// TwinCAT 3 PLC project Plc
// ProgramVersion: 3.1.4024.0
// libraries:
//   Tc2_Standard, * (Beckhoff Automation GmbH)
//   Tc2_System, * (Beckhoff Automation GmbH)
//   Tc3_Module, * (Beckhoff Automation GmbH)
//   VisuDialogs, * (System)
// project tree:
//   / Gestore di visualizzazione.TcVMO (not stored), GlobalTextList.TcGTLO, ImagePool.TcIPO (not stored), PlcTask.TcTTO, VisuTask.TcTTO
//   GVLs/ GVL.TcGVL (not stored)
//   POUs/ MAIN.TcPOU, VISU.TcPOU
//   VISUs/ Visualization.TcVIS
// real-time tasks:
//   TASK PlcTask: cycle T#10ms, priority 20, ADS port 350
//   TASK VisuTask: cycle T#100000us, priority 60, ADS port 351

CONFIGURATION Plc
    RESOURCE PLC ON TwinCAT3
        TASK PlcTask(INTERVAL := T#10ms, PRIORITY := 20);
        TASK VisuTask(INTERVAL := T#100000us, PRIORITY := 60);
        PROGRAM MAIN WITH PlcTask : MAIN;
    END_RESOURCE
END_CONFIGURATION

// ---- POUs/MAIN.TcPOU
PROGRAM MAIN
VAR
	StopRichiesto: BOOL;
	Anomalia: BOOL;
	Emergenza: BOOL;
	Funzione: BOOL;
	Smistamento: BOOL;
	Rotazione: BOOL;
	AttivaMicroRulli: BOOL;
	FineSmistamento: BOOL;
	FinePesatura: BOOL;
	RuotaOrigine: BOOL;
	PesoMin5: BOOL;
	PesoMag10: BOOL;
	PesoIntermedio: BOOL;
	ProsciuttoSmistato: BOOL;
	ProsciuttiTotali: UINT;
	ProsciuttiCommerciabili: UINT;
	PercentualeProsciuttiCommerciabili: UINT;
	//Timer
	TON_PS1: TON;
	TON_Pesatura: TON;
	TON_MicroRulli: TON;
	TON_Min5: TON;
	TON_Mag10: TON;
	TON_Intermedi: TON;
	//Counter
	CTU_Min5: CTU;
	CTU_Mag10: CTU;
	CTU_Intermedi: CTU;
END_VAR

GestionePulsanti();
GestioneMotori();
GestionePesatura();
GestioneRotazione();
GestioneSmistamento();
GestioneConteggio();

ACTION GestioneConteggio:
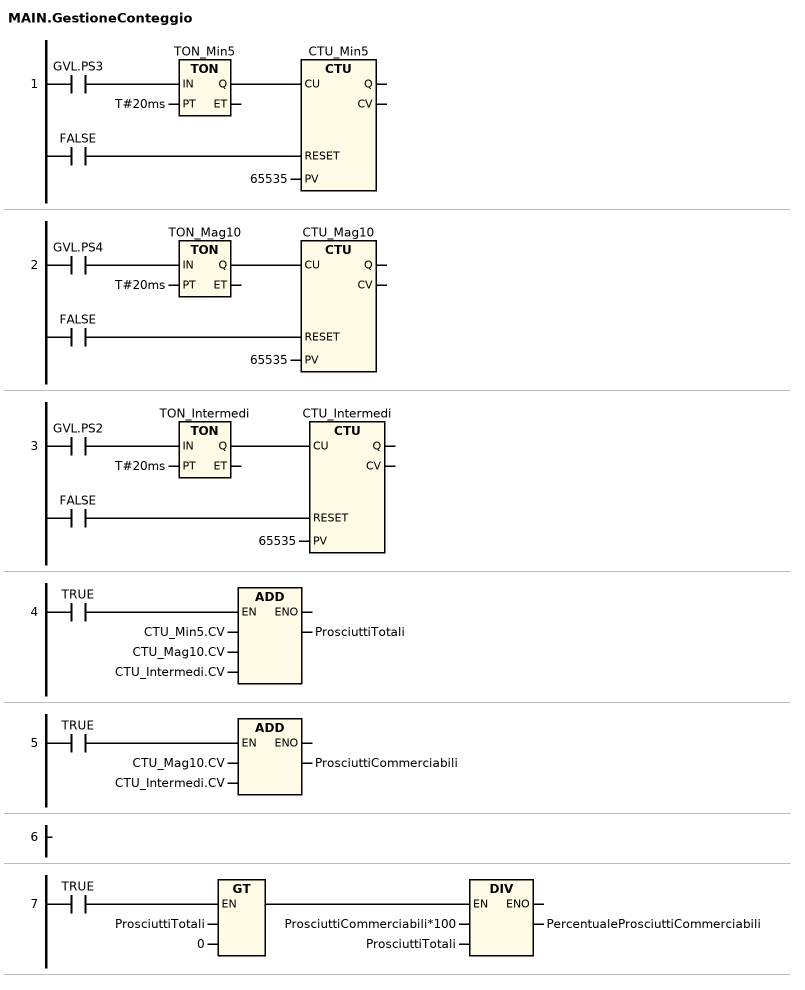
// NETWORK 1
TON_Min5(IN := GVL.PS3, PT := T#20ms); // TON
CTU_Min5(CU := TON_Min5.Q, RESET := FALSE, PV := 65535); // CTU

// NETWORK 2
TON_Mag10(IN := GVL.PS4, PT := T#20ms); // TON
CTU_Mag10(CU := TON_Mag10.Q, RESET := FALSE, PV := 65535); // CTU

// NETWORK 3
TON_Intermedi(IN := GVL.PS2, PT := T#20ms); // TON
CTU_Intermedi(CU := TON_Intermedi.Q, RESET := FALSE, PV := 65535); // CTU

// NETWORK 4
ProsciuttiTotali := CTU_Min5.CV + CTU_Mag10.CV + CTU_Intermedi.CV;

// NETWORK 5
ProsciuttiCommerciabili := CTU_Mag10.CV + CTU_Intermedi.CV;

// NETWORK 6

// NETWORK 7
IF ProsciuttiTotali > 0 THEN
    PercentualeProsciuttiCommerciabili := (ProsciuttiCommerciabili*100) / ProsciuttiTotali;
END_IF
END_ACTION

ACTION GestioneMotori:
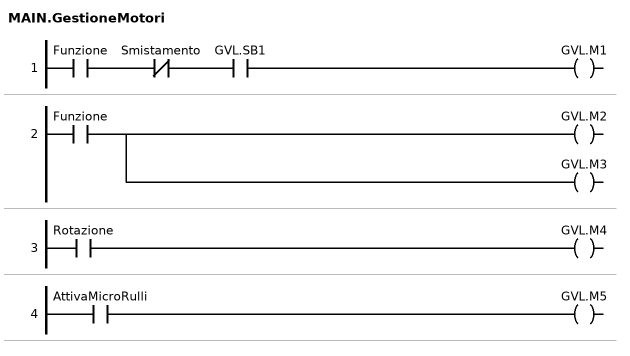
// NETWORK 1
GVL.M1 := Funzione AND NOT Smistamento AND GVL.SB1;

// NETWORK 2
GVL.M2 := Funzione;
GVL.M3 := Funzione;

// NETWORK 3
GVL.M4 := Rotazione;

// NETWORK 4
GVL.M5 := AttivaMicroRulli;
END_ACTION

ACTION GestionePesatura:
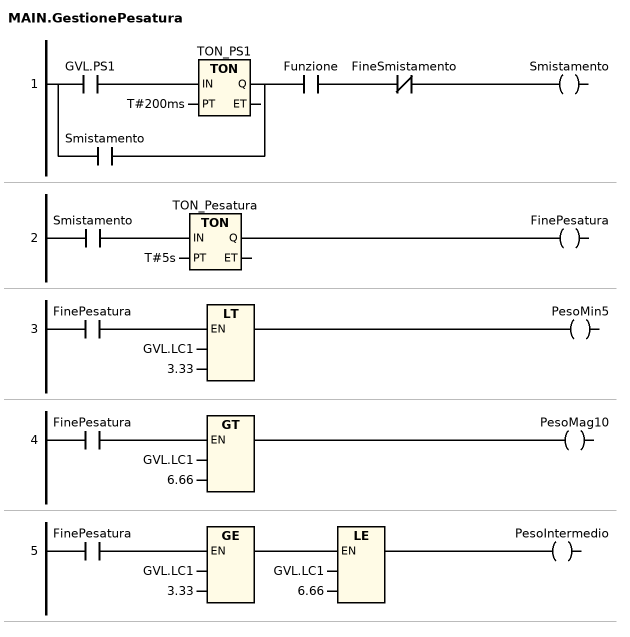
// NETWORK 1
TON_PS1(IN := GVL.PS1, PT := T#200ms); // TON
Smistamento := (TON_PS1.Q OR Smistamento) AND Funzione AND NOT FineSmistamento;

// NETWORK 2
TON_Pesatura(IN := Smistamento, PT := T#5s); // TON
FinePesatura := TON_Pesatura.Q;

// NETWORK 3
PesoMin5 := FinePesatura AND GVL.LC1 < 3.33;

// NETWORK 4
PesoMag10 := FinePesatura AND GVL.LC1 > 6.66;

// NETWORK 5
PesoIntermedio := FinePesatura AND GVL.LC1 >= 3.33 AND GVL.LC1 <= 6.66;
END_ACTION

ACTION GestionePulsanti:
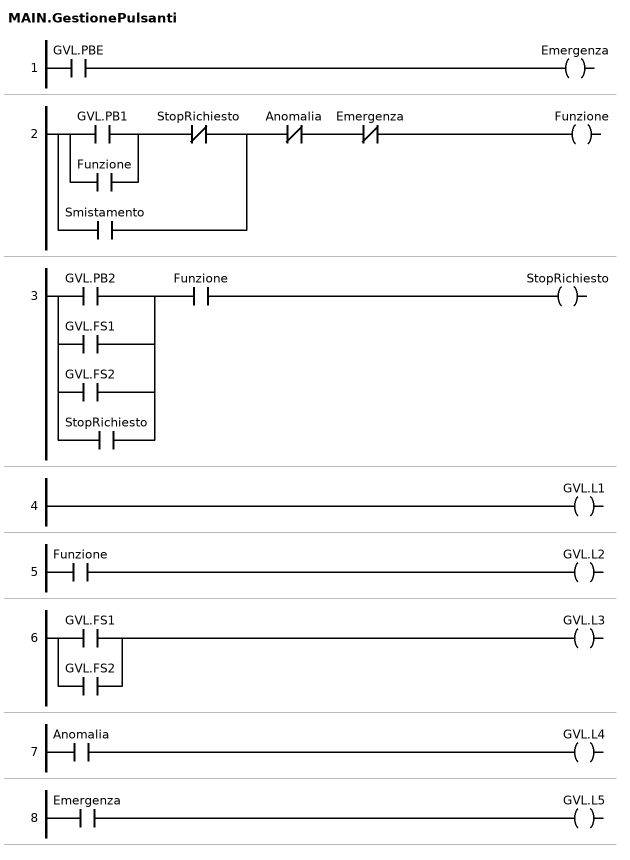
// NETWORK 1
Emergenza := GVL.PBE;

// NETWORK 2
Funzione := ((GVL.PB1 OR Funzione) AND NOT StopRichiesto OR Smistamento) AND NOT Anomalia AND NOT Emergenza;

// NETWORK 3
StopRichiesto := (GVL.PB2 OR GVL.FS1 OR GVL.FS2 OR StopRichiesto) AND Funzione;

// NETWORK 4
GVL.L1 := TRUE;

// NETWORK 5
GVL.L2 := Funzione;

// NETWORK 6
GVL.L3 := GVL.FS1 OR GVL.FS2;

// NETWORK 7
GVL.L4 := Anomalia;

// NETWORK 8
GVL.L5 := Emergenza;
END_ACTION

ACTION GestioneRotazione:
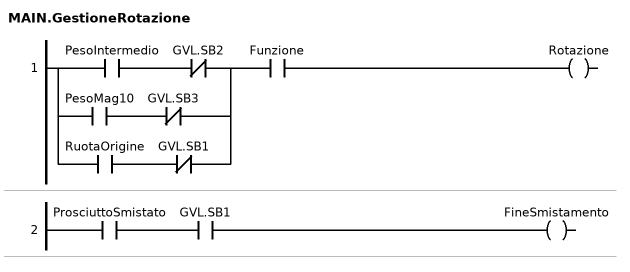
// NETWORK 1
Rotazione := (PesoIntermedio AND NOT GVL.SB2 OR PesoMag10 AND NOT GVL.SB3 OR RuotaOrigine AND NOT GVL.SB1) AND Funzione;

// NETWORK 2
FineSmistamento := ProsciuttoSmistato AND GVL.SB1;
END_ACTION

ACTION GestioneSmistamento:
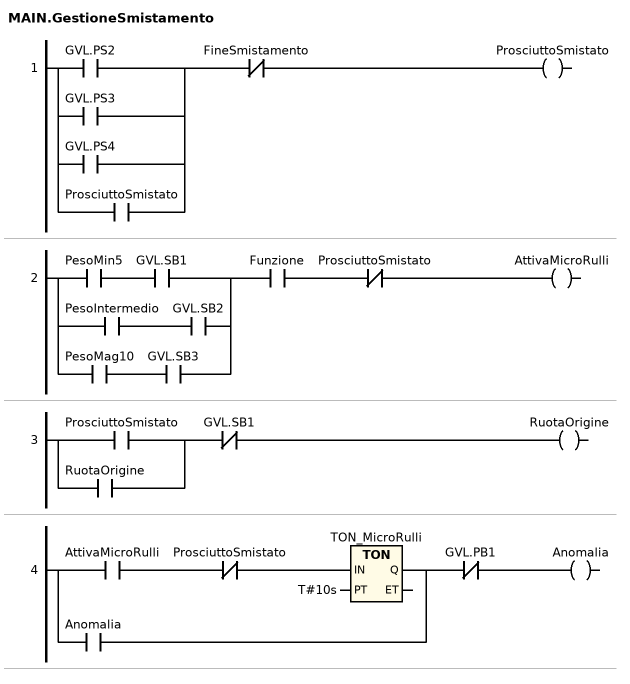
// NETWORK 1
ProsciuttoSmistato := (GVL.PS2 OR GVL.PS3 OR GVL.PS4 OR ProsciuttoSmistato) AND NOT FineSmistamento;

// NETWORK 2
AttivaMicroRulli := (PesoMin5 AND GVL.SB1 OR PesoIntermedio AND GVL.SB2 OR PesoMag10 AND GVL.SB3) AND Funzione AND NOT ProsciuttoSmistato;

// NETWORK 3
RuotaOrigine := (ProsciuttoSmistato OR RuotaOrigine) AND NOT GVL.SB1;

// NETWORK 4
TON_MicroRulli(IN := AttivaMicroRulli AND NOT ProsciuttoSmistato, PT := T#10s); // TON
Anomalia := (TON_MicroRulli.Q OR Anomalia) AND NOT GVL.PB1;
END_ACTION

END_PROGRAM

// ---- POUs/VISU.TcPOU
PROGRAM VISU
VAR
	posizioneProsciutto: INT;
	posizioneProsciuttoY: INT;
	rotazionePiattaforma: INT;
	prosciuttoVisibile: BOOL;
	Random: DRAND;
	PB1Trig: R_TRIG;
	SmistamentoTrig: F_TRIG;
END_VAR

Random(Seed:= 100); //Numero casuale
PB1Trig(CLK := GVL.PB1); //Fronte di salita del pulsante
SmistamentoTrig(CLK := MAIN.Smistamento); //Indica quando termina uno smistamento

//Reset posizione alla fine dello smistamento o alla pressione di Start
IF PB1Trig.Q OR SmistamentoTrig.Q THEN
	GVL.LC1 := Random.Num * 10;
	prosciuttoVisibile := TRUE;
	posizioneProsciutto := 0;
	posizioneProsciuttoY := 0;
	rotazionePiattaforma := 0;
	GVL.PS1 := 0;
END_IF

IF GVL.M1 THEN
	posizioneProsciutto := posizioneProsciutto +2;
END_IF

IF GVL.M5 AND rotazionePiattaforma = 0 THEN
	posizioneProsciutto := posizioneProsciutto +4;
END_IF

IF GVL.M5 AND rotazionePiattaforma = 90 THEN
	posizioneProsciuttoY := posizioneProsciuttoY +2;
END_IF

IF GVL.M5 AND rotazionePiattaforma = 270 THEN
	posizioneProsciuttoY := posizioneProsciuttoY -2;
END_IF

IF posizioneProsciutto >= 160 AND NOT MAIN.Smistamento THEN
	GVL.PS1 := TRUE;
ELSE
	GVL.PS1 := FALSE;
END_IF

IF posizioneProsciutto >= 350 THEN
	GVL.PS3 := TRUE;
	prosciuttoVisibile:= FALSE;
ELSE
	GVL.PS3 := FALSE;
END_IF

IF posizioneProsciuttoY >= 200 THEN
	GVL.PS2 := TRUE;
	prosciuttoVisibile:= FALSE;
ELSE
	GVL.PS2 := FALSE;
END_IF

IF posizioneProsciuttoY <= -200 THEN
	GVL.PS4 := TRUE;
	prosciuttoVisibile:= FALSE;
ELSE
	GVL.PS4 := FALSE;
END_IF



IF GVL.M4 THEN
	rotazionePiattaforma := rotazionePiattaforma +2;
	IF rotazionePiattaforma = 360 THEN
		rotazionePiattaforma := 0;
	END_IF
END_IF

CASE rotazionePiattaforma OF
	0:
		GVL.SB1 := TRUE;
		GVL.SB2 := FALSE;
		GVL.SB3 := FALSE;
	90:
		GVL.SB1 := FALSE;
		GVL.SB2 := TRUE;
		GVL.SB3 := FALSE;
	270:
		GVL.SB1 := FALSE;
		GVL.SB2 := FALSE;
		GVL.SB3 := TRUE;
	ELSE
		GVL.SB1 := FALSE;
		GVL.SB2 := FALSE;
		GVL.SB3 := FALSE;
END_CASE

END_PROGRAM

// ---- GlobalTextList.TcGTLO
TEXTLIST GlobalTextList
  628 = '%d'
  216 = '%f'
  68 = 'Emergenza'
  801 = 'FS1'
  524 = 'FS2'
  765 = 'LC1'
  869 = 'M1'
  802 = 'M2'
  115 = 'M3'
  287 = 'M4'
  498 = 'M5'
  501 = 'Percentuale prosciutti commerciabili: %d'
  820 = 'Percentuale prosciutti commerciabili:%d'
  388 = 'PS1'
  310 = 'PS2'
  806 = 'PS3'
  525 = 'PS4'
  656 = 'SB1'
  665 = 'SB2'
  112 = 'SB3'
  871 = 'Start'
  275 = 'Stop'
END_TEXTLIST

// ---- VISUs/Visualization.TcVIS
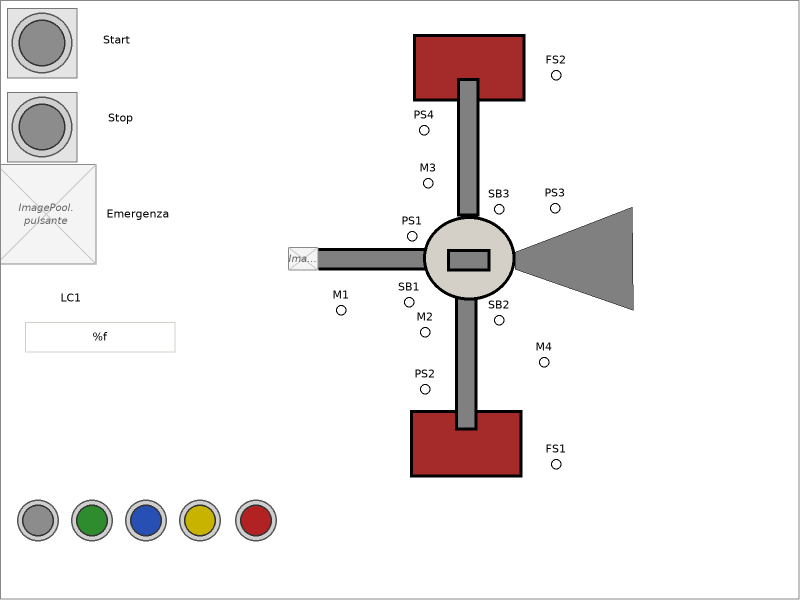
VISUALIZATION Visualization  // 800x600
    Rectangle (473,-103 67x112), angle 270
    Rectangle (470,273 67x112), angle 270
    PushSwitch (7,8 70x70), variable: GVL.PB1, behaviour: TAP, style: Switch-PushSwitch-Gray
    Label (89,25 55x30), "Start"
    PushSwitch (7,92 70x70), variable: GVL.PB2, behaviour: TAP, style: Switch-PushSwitch-Gray
    Label (88,103 65x30), "Stop"
    Label (93,199 90x30), "Emergenza"
    Rectangle (289,248 138x22)
    Rectangle (304,201 138x22), angle 90
    Rectangle (302,415 138x22), angle 90
    Ellipse (423,216 92x84)
    Polygon (515,252) (557,236) (632,207) (633,310) (515,269)
    Ellipse (407,231 10x10), colour toggle: GVL.PS1
        tap GVL.PS1
    Label (388,215 48x12), "PS1"
    Lamp1 (14,496 48x49), variable: GVL.L1, style: Lamp-Lamp1-Gray
    Lamp1 (68,496 48x49), variable: GVL.L2, style: Lamp-Lamp1-Green
    Lamp1 (122,496 48x49), variable: GVL.L3, style: Lamp-Lamp1-Blue
    Lamp1 (176,496 48x49), variable: GVL.L4, style: Lamp-Lamp1-Yellow
    Lamp1 (232,496 48x49), variable: GVL.L5, style: Lamp-Lamp1-Red
    Ellipse (551,459 10x10), colour toggle: GVL.FS1
        toggle GVL.FS1
    Label (532,443 48x12), "FS1"
    Ellipse (551,70 10x10), colour toggle: GVL.FS2
        toggle GVL.FS2
    Label (532,54 48x12), "FS2"
    Ellipse (420,384 10x10), colour toggle: GVL.PS2
        tap GVL.PS2
    Label (401,368 48x12), "PS2"
    Ellipse (550,203 10x10), colour toggle: GVL.PS3
        tap GVL.PS3
    Label (531,187 48x12), "PS3"
    Ellipse (419,125 10x10), colour toggle: GVL.PS4
        tap GVL.PS4
    Label (400,109 48x12), "PS4"
    Label (317,289 48x12), "M1"
    Ellipse (336,305 10x10), colour toggle: GVL.M1
    Label (401,311 48x12), "M2"
    Ellipse (420,327 10x10), colour toggle: GVL.M2
    Label (404,162 48x12), "M3"
    Ellipse (423,178 10x10), colour toggle: GVL.M3
    Label (520,341 48x12), "M4"
    Ellipse (539,357 10x10), colour toggle: GVL.M4
    Textfield (25,322 150x30), "%f", text variable: GVL.LC1
        OnMouseClick: write GVL.LC1 via VisuDialogs.Numpad, min 0, max 10
    Label (26,283 90x30), "LC1"
    Ellipse (494,315 10x10), colour toggle: GVL.SB2
        toggle GVL.SB2
    Label (475,299 48x12), "SB2"
    Label (475,188 48x12), "SB3"
    Ellipse (494,204 10x10), colour toggle: GVL.SB3
        toggle GVL.SB3
    Label (385,281 48x12), "SB1"
    Ellipse (404,297 10x10), colour toggle: GVL.SB1
        toggle GVL.SB1
    Rectangle (447,249 43x22), angle 180, colour toggle: GVL.M5
        p2858320360: VISU.rotazionePiattaforma
    Image (288,247 30x23), invisible if: NOT VISU.prosciuttoVisibile, image: ImagePool.ham
        p3560616238: VISU.posizioneProsciutto
        p2858320360: VISU.rotazionePiattaforma
        p2738717112: VISU.posizioneProsciuttoY
    Image (-4,164 100x100), image: ImagePool.pulsante
        OnMouseClick: toggle GVL.PBE
END_VISUALIZATION
